// TIA Portal V16 export
// export: Created 2021-07-12T14:47:19.9182028Z, ExportSetting WithDefaults, DisplayName Totally Integrated Automation Portal, DisplayVersion V16, DisplayName TIA Portal Version Control Interface, DisplayVersion V16, DisplayName TIA Portal Openness, DisplayVersion V16, DisplayName STEP 7 Professional, DisplayVersion V16, DisplayName STEP 7 Safety, DisplayVersion V16, DisplayName WinCC Professional, DisplayVersion V16
TYPE "LSimaHydTO_typeMeasurementQOutput"
TITLE = LSimaHydTO_typeMeasurementQOutput
// Structure to define the manipulated variable
// stored: IsFailsafeCompliant false
   STRUCT
      enableMeasurement { S7_SetPoint := 'True'} : Bool := TRUE;   // Enables measurement in this direction
      maxVelocity { S7_SetPoint := 'True'} : Real := 500.0;   // Velocity limit in this direction
      setpointForMovement { S7_SetPoint := 'True'} : Real := 40.0;   // Substitute value for movements if a measurement is not active [%]
      ramp { S7_SetPoint := 'True'} : Real := 100.0;   // manipulated variable – increase/decrease [%/s]
      minQOutputValue { S7_SetPoint := 'True'} : Real;   // start measurement with this value
      fineRange { S7_SetPoint := 'True'} : "LSimaHydTO_typeMeasurementQOutputRange";   // measurement in the fine area
      coarseRange { S7_SetPoint := 'True'} : "LSimaHydTO_typeMeasurementQOutputRange";   // measurement in the coarse area
   END_STRUCT;
   // fineRange.maxQOutputValue := 40.0;
   // fineRange.numberOfPoints := 10;
   // coarseRange.maxQOutputValue := 100.0;
   // coarseRange.numberOfPoints := 10;
END_TYPE
